{attribute 'linkalways'} 
{attribute 'no_explicit_call' := 'This FB is a CLASS and must be accessed using methods or properties'}
{attribute 'enable_dynamic_creation'}
FUNCTION_BLOCK FINAL LT_UINT EXTENDS Node
VAR
	in1 : _UINT(0);
	in2 : _UINT(0);
	out : _BOOL(FALSE);
END_VAR

METHOD PUBLIC Clone : I_Node
VAR
	pNode : POINTER TO LT_UINT;
END_VAR
pNode := __NEW(LT_UINT);
Clone := pNode^;
END_METHOD

METHOD FB_init : BOOL
VAR_INPUT
	bInitRetains : BOOL; // if TRUE, the retain variables are initialized (warm start / cold start)
	bInCopyCode : BOOL;  // if TRUE, the instance afterwards gets moved into the copy code (online change)
END_VAR
AddInput('in1',THIS^.in1);
AddInput('in2',THIS^.in2);
AddOutput('out', THIS^.out);
END_METHOD

METHOD PROTECTED OnExecute
VAR
END_VAR
out.Value := in1.Value < in2.Value;
END_METHOD

END_FUNCTION_BLOCK

(* stored: Version 1.1.0.1, ProductVersion 3.1.4024.15
   POU LT_UINT: Id {a0fe0613-13f4-4539-b50d-e9d3756aa25c}, SpecialFunc None
   Folder Constructor: Id {9f4a6108-f60c-48a2-83c1-7a247774de52}
   Method Clone: Id {fea0387e-1337-4a03-a982-8bce72255486}
   Method FB_init: Id {1d0c6b07-6298-4dca-bebf-bcda75c12e53}
   Method OnExecute: Id {c78a0482-7b78-4676-9077-cede6f45bd6d} *)
